// TIA Portal V17 export
// export: Created 2024-08-09T12:53:16.4149239Z, ExportSetting WithDefaults, DisplayName Totally Integrated Automation Portal, DisplayVersion V17 Update 7, DisplayName TIA Portal Openness, DisplayVersion V17 Update 7, DisplayName TIA Portal Version Control Interface, DisplayVersion V17, DisplayName STEP 7 Professional, DisplayVersion V17 Update 7, DisplayName STEP 7 Safety, DisplayVersion V17 Update 6, DisplayName WinCC Professional, DisplayVersion V17 Update 7
TYPE "utSql4SiemensInterface"
// stored: IsFailsafeCompliant false
   STRUCT
      Observer : Struct
         Dial_Def { S7_SetPoint := 'True'} : "S_DIALOG_DEF";
         _Etp { ExternalAccessible := 'False'; ExternalVisible := 'False'; ExternalWritable := 'False'} : SInt;
         _EtpPrec { ExternalAccessible := 'False'; ExternalVisible := 'False'; ExternalWritable := 'False'} : SInt;
         _EtpMemo { ExternalAccessible := 'False'; ExternalVisible := 'False'; ExternalWritable := 'False'} : SInt;
         _TpsPicke { ExternalAccessible := 'False'; ExternalVisible := 'False'; ExternalWritable := 'False'} : Date_And_Time;
         xTimeout { ExternalVisible := 'False'} : Bool := FALSE;
      END_STRUCT;
      xExecute : Bool;
      xHoldConnection : Bool;
      xUseMrpParameter : Bool := true;
      diRequestDataSize : DInt := 0;
      CutString : DInt := 600;
      abRequestData : Array[0..10000] of Byte;
      diResponseDataSize : DInt := 0;
      abResponseData : Array[0..10000] of Byte;
      cdiResponseReturnParamSize : DInt := 50;
      adiResponseReturnParam : Array[0..49] of Struct
         diOffset : DInt;
         iLength : Int;
      END_STRUCT;
      cdiResponseRowSize : DInt := 50;
      cdiResponseColumnSize : DInt := 20;
      adiResponseColumnName : Array[0..19] of Struct
         diOffset : DInt;
         iLength : Int;
      END_STRUCT;
      adiResponseData : Array[0..49, 0..19] of Struct
         diOffset : DInt;
         iLength : Int;
      END_STRUCT;
      cdiResponseMaxStringSize : DInt := 6000;
      xReady : Bool;
      xBusy : Bool;
      xDone : Bool;
      xError : Bool;
      diResultState : DInt;
      diResultReturnParams : DInt;
      diResultRows : DInt;
      diResultColumns : DInt;
   END_STRUCT;
END_TYPE
